PROGRAM Fahrauftrag
VAR
	//State machine
	sStart : BOOL := TRUE;
	s0,s1a,s1b,s2,s3,s4,s5,s6a,s6b,s7,s8,s9,s10,s11a,s11b,s12,s13,s14,s15,s16,s17,s18,s19,s20,s21a,s21b,s22,s23,s24,s25,s26a,s26b,s27,s28,s29,s30,s31: BOOL := FALSE;
	sk0, sk1, sk2, sk3, sk4, sk10, sk20, sk21, sk22, sk23, sk24, sk25, sk26, sk27, sk28, sk29, sk30, sk31 : BOOL := FALSE; //States von Kollision
	
	AStar : AStar;										//A-Stern Algorithmus
	readAssigment: ReadAssigment;						//Auswertung des Auftrags
	TrajectoryController: TrajectoryControl;			//Schnittstelle zu GW3
	
	wayPointList : ARRAY[0..100] OF RobotPoseSimple;	//Wegpunktliste
	actualCamX, actualCamY : LREAL;						//letzte Kameradaten ungleich 0
	lastRelevantStateForCollision : STRING(5);			//letzter State für Rückfall bei Kollision
	
	//Schnittstelle zum MQTT_PRG
	FeedbackToGW1 AT%Q*: STRING(50);		//Feedback/Status des Roboters an GW1
	resetVar, resetGoBack AT%Q*: BOOL;					//messages von MQTT zurücksetzen
	RoboNmbToGoBack AT%Q* : INT;
	Auftrag AT%I*: Auftrag;					//Auftrag von GW1
	StatusFromGW1 AT%I*: STRING(50);		//Status von GW1
	goBack AT%I* : BOOL;					//zurückfahren auf Befehl von anderem HAWino
	reset AT%I* : BOOL;						//Fahrauftrag und GW3 zurücksetzen auf Befehl von GW1
	
	//Schnittstelle zu A*-Algorithmus
	EndNode : INT;							//letzter Knoten
	xEndvalue : LREAL;						//Ziel xKoordinate
	xRobotStartposition : LREAL;			//aktuelle xKoordinate
	yEndvalue : LREAL;						//Ziel yKoordinate
	yRobotStartposition : LREAL;			//aktuelle yKoordinate
	xPointList : ARRAY[0..100] OF LREAL;	//xKoordinatenliste
	yPointList : ARRAY[0..100] OF LREAL;	//yKoordinatenliste
	finished_ASearch : BOOL;	 			//Variable, dass Algorithmus fertig
	i: INT;									//Laufvariable zum Übertragen der x und y Koordinaten in die Wegpunktliste
	zeile: INT;								//Arrayindex, wo Wegpunktliste zuende
	
	//Kollision
	collision AT%I*: ARRAY[0..4] OF BOOL;		//Collision wurde erkannt
	lastCollision: ARRAY [0..4] OF BOOL;		//letzte Collision gespeichert
	collisionFree, collisionSolutionWorking : BOOL;				//keine Kollision aktuell
	removeNodeCollision : ARRAY[1..11] OF INT;	//Nodes die durch anderen HAWino blockiert
	todo : STRING(10);							//Aufgabe von diesem HAWino bei Kollision (fahren oder warten)
	firstTime: BOOL := TRUE;	
	timerCollision : TON;						//Zeit die bei Kollision gewartet wird, bevor Reaktion folgt
	otherRobo : ARRAY[0..4] OF INT;				//andere HAWinos, die an Kollision beteilgit
	otherRoboAtStation, otherRoboAtStop, thisRoboAtStation, drivingAtStation, newCollision : BOOL;			//anderer beteiligter HAWino ist im Stationsbereich
	
	//error
	noCamera, AStarFailed, error, test : BOOL;
	resetTimer : TON;
END_VAR

timerCollision();
resetTimer();
errorTest();

collisionFree := NOT collision[Var_HAWIno.Robot_Number];

//neue Kollision angekommen oder noch alte?
//IF lastCollision[1] <> collision[1] OR lastCollision[2] <> collision[2] OR lastCollision[3] <> collision[3] OR lastCollision[4] <> collision[4] OR collision[0] THEN
//	IF collision[Var_HAWIno.Robot_Number] THEN
//		TrajectoryController.xBoEnable := FALSE;
//		CollisionSolution();
//		timerCollision.IN := TRUE;
//		timerCollision.PT := T#2S;
//	END_IF
//	lastCollision := collision;
//LSIF (todo = 'Warten' AND collisionFree) OR timerCollision.Q THEN
//	CollisionSolution();	
//	timerCollision.IN := FALSE;
//ELSIF (goBack AND NOT resetGoBack) OR (otherRoboAtStation AND todo = 'Warten') THEN
//	drivingBack();
//	todo := 'Warten';
//ELSIF resetGoBack AND NOT goBack THEN
//	resetGoBack := FALSE;
//END_IF

IF lastCollision[1] <> collision[1] OR lastCollision[2] <> collision[2] OR lastCollision[3] <> collision[3] OR lastCollision[4] <> collision[4] OR collision[0] THEN
	newCollision := TRUE;
	lastCollision := collision;
END_IF

IF collision[Var_HAWIno.Robot_Number] AND newCollision THEN
	TrajectoryController.xBoEnable := FALSE;
	IF NOT collisionSolutionWorking THEN
		sk0 := TRUE;
	END_IF
	CollisionsSolution_new();
	newCollision := FALSE;
	timerCollision.IN := TRUE;
	timerCollision.PT := T#2S;
ELSIF collisionSolutionWorking THEN
	CollisionsSolution_new();
END_IF

//Camera damit immer Daten da
IF camera.cameraData.robotPositionArray[Var_HAWIno.Robot_Number].x <> 0 AND camera.cameraData.robotPositionArray[Var_HAWIno.Robot_Number].y <> 0 THEN
	actualCamX := camera.cameraData.robotPositionArray[Var_HAWIno.Robot_Number].x;
	actualCamY := camera.cameraData.robotPositionArray[Var_HAWIno.Robot_Number].y;
END_IF

////////////////////////////////////////////////////////StateMaschine/////////////////////////////////////////////////

//Init
IF sStart AND NOT s0 THEN
	lastRelevantStateForCollision := 's0';
	sStart := 0; s0 := 1;
	//	RückmeldungGW1 Verfügbar
	FeedbackToGW1 := 'Verfuegbar';
	resetVar := FALSE;
	TrajectoryController.xBoReset := FALSE;
END_IF

//////////////////////////////////////////////////////////////////////////////////////////////////////////////
//////////////////////////////////FAHRAUFTRAG/////////////////////////////////////////////////////////////////
//////////////////////////////////////////////////////////////////////////////////////////////////////////////

//	Warten auf Auftrag
IF s0 AND NOT s1a AND Auftrag.Art = 'Fahrauftrag' THEN
	s0 := 0; s1a := 1;
	lastRelevantStateForCollision := 's1a';
	//	RückmeldugGW1 Auftrag angenommen setzt
	FeedbackToGW1 := 'Auftrag angenommen';
	//Auftrag auswerten
	readAssigment(assigment:= Auftrag);
	EndNode := readAssigment.endNodePickup;															
	xEndvalue := readAssigment.pickupLocation.x;
	yEndvalue := readAssigment.pickupLocation.y;
	xRobotStartposition := camera.cameraData.robotPositionArray[Var_HAWIno.Robot_Number].x;
	yRobotStartposition := camera.cameraData.robotPositionArray[Var_HAWIno.Robot_Number].y;	
END_IF

IF s1a AND NOT s1b AND xRobotStartposition <> 0 AND yRobotStartposition <> 0 THEN
	s1a := 0; s1b := 1;
	AStar(xRobotActual := xRobotStartposition, yRobotActual := yRobotStartposition, xEnd := xEndvalue, yEnd := yEndvalue, endNode := EndNode, blockedNodes := removeNodeCollision);
	finished_ASearch := AStar.finishedASearch;
	xPointList := AStar.xCoordinates;
	yPointList := AStar.yCoordinates;
	ZEROS_INT(removeNodeCollision);
ELSIF s1a AND NOT s1b THEN
	xRobotStartposition := actualCamX;
	yRobotStartposition := actualCamY;
END_IF

//Bahnplanung
IF s1b AND NOT s2 AND finished_ASearch THEN
	ZEROS_RobotPoseSimple(wayPointList);
	FOR i := 0 TO 100 BY 1 DO
 		wayPointList[i] := ToRobotPoseSimple(x:= xPointList[i], y:= yPointList[i], theta:= -1);
		IF xPointList[i] = 0 THEN
			zeile := i;
			EXIT;
		END_IF
	END_FOR
	wayPointList[zeile] := readAssigment.pickupLocation;
	wayPointList[zeile+1] := ToRobotPoseSimple(x := -1, y := -1, theta := -1);
	//wayPointList[zeile+2] := readAssigment.lastPointsToPickup[2];
	TrajectoryController.setWaypointList(waypointList);
	trajectoryController.newWaypointListAvailable := TRUE;
	s1b := 0; s2 := 1;
END_IF

///////////////////////////////////////////////FahrtZumAbholort///////////////////////////////////////////////////

// 	RückmeldungGW3 Wegpunkte erhalten abwarten
IF s2 AND NOT s3 AND trajectoryController.yControllerState = ControllerState.setTrajectory THEN
	s2 := 0; s3 := 1;
	trajectoryController.newWaypointListAvailable := FALSE;
END_IF

// 	RückmeldungGW3 ready abwarten
IF s3 AND NOT s4 AND trajectoryController.yControllerState = ControllerState.ready THEN
	s3 := 0; s4 := 1;
	trajectoryController.xBoEnable := TRUE;
END_IF
	
//	RückmeldungGW3 Fahrt abwarten
IF s4 AND NOT s5 AND trajectoryController.yControllerState = ControllerState.driving THEN
	s4 := 0; s5 := 1;
	//	RückmeldungGW1 Auf Anfahrt setzen
	FeedbackToGW1 := 'Auf Anfahrt';
END_IF

//	RückmeldungGW3 am Ziel abwarten
IF s5 AND NOT s6a AND trajectoryController.yBoArrivedAtDestination THEN
	s5 := 0; s6a := 1;
	lastRelevantStateForCollision := 's6a';
	trajectoryController.xBoEnable := FALSE;
	//	Greifersteuerung
	Gripper.closeGripperCommand := TRUE;
END_IF
												// hier könnte noch slider und Lichtschranke abgefragt werden zur Sicherheit
IF s6a AND NOT s6b AND NOT Gripper.partGripped THEN
	s6a := 0; s6b := 1;	
	//	RückmeldungGW1 Teil aufgenommen setzen
	FeedbackToGW1 := 'Teil aufgenommen';
	//	Fahrauftrag zu Lesekopf
	ZEROS_RobotPoseSimple(wayPointList);
	wayPointList := readAssigment.pointsFromSlotToReader;
	TrajectoryController.setWaypointList(wayPointList);
	trajectoryController.newWaypointListAvailable := TRUE;
ELSIF s6a AND NOT s6b AND Gripper.partGripped THEN
	Gripper.closeGripperCommand := FALSE;
	ZEROS_RobotPoseSimple(wayPointList);										//test, sonst für alle
	wayPointList[0] := ToRobotPoseSimple(x := readAssigment.pickupLocation.x - 100, y := readAssigment.pickupLocation.y, theta := readAssigment.pickupLocation.theta);
	wayPointList[1] := readAssigment.pickupLocation;
	wayPointList[2] := ToRobotPoseSimple(x := -1, y := -1, theta := -1);
	TrajectoryController.setWaypointList(waypointList);
	trajectoryController.newWaypointListAvailable := TRUE;
	s6a := 0; s2 := 1;
END_IF


/////////////////////////////////////////////////////FahrtZumLesekopf/////////////////////////////////////////////////////////

// 	RückmeldungGW3 Wegpunkte erhalten abwarten
IF s6b AND NOT s7 AND trajectoryController.yControllerState = ControllerState.setTrajectory AND gripper.state = CoreGripperControlState.Open THEN
	s6b := 0; s7 := 1;
	trajectoryController.newWaypointListAvailable := FALSE;
END_IF

// 	RückmeldungGW3 ready abwarten
IF s7 AND NOT s8 AND trajectoryController.yControllerState = ControllerState.ready THEN
	s7 := 0; s8 := 1;
	trajectoryController.xBoEnable := TRUE;
END_IF
	
//	RückmeldungGW3 Fahrt abwarten
IF s8 AND NOT s9 AND trajectoryController.yControllerState = ControllerState.driving THEN
	s8 := 0; s9 := 1;
END_IF

//	RückmeldungGW3 am Ziel abwarten
IF s9 AND NOT s10 AND trajectoryController.yBoArrivedAtDestination THEN
	s9 := 0; s10 := 1;
	lastRelevantStateForCollision := 's10';
	trajectoryController.xBoEnable := FALSE;
	//	RückmeldungGW1 Abmeldung
	FeedbackToGW1 := 'Abmeldung';
END_IF

//	Warten auf Werkstück ausgelesen
IF s10 AND NOT s11a AND StatusFromGW1 = 'WerkstueckAusgelesen' THEN
	s10 := 0; s11a := 1;
	lastRelevantStateForCollision := 's11a';
	resetVar := TRUE;
	
	//Auftrag auswerten
	EndNode   := readAssigment.endNodeStorage;																	
	xEndvalue := readAssigment.storageLocation.x;
	yEndvalue := readAssigment.storageLocation.y;
	yRobotStartposition := camera.cameraData.robotPositionArray[Var_HAWIno.Robot_Number].y;	
	xRobotStartposition := camera.cameraData.robotPositionArray[Var_HAWIno.Robot_Number].x;
	//IF readAssigment.assigment.AbholTasche < 3 THEN
	//	xRobotStartposition := camera.cameraData.robotPositionArray[Var_HAWIno.Robot_Number].x - 200;
	//ELSE
	//	xRobotStartposition := camera.cameraData.robotPositionArray[Var_HAWIno.Robot_Number].x + 200;
	//END_IF
END_IF

IF s11a AND NOT s11b AND xRobotStartposition <> 0 AND yRobotStartposition <> 0 THEN
	s11a := 0; s11b := 1;
	AStar(xRobotActual := xRobotStartposition, yRobotActual := yRobotStartposition, xEnd := xEndvalue, yEnd := yEndvalue, endNode := EndNode, blockedNodes := removeNodeCollision);
	finished_ASearch := AStar.finishedASearch;
	xPointList := AStar.xCoordinates;
	yPointList := AStar.yCoordinates;
	ZEROS_INT(removeNodeCollision);
ELSIF s11a AND NOT s11b THEN
	//IF readAssigment.assigment.AbholTasche < 3 THEN	
	//	xRobotStartposition := actualCamX - 200;
	//ELSE
	//	xRobotStartposition := actualCamX + 200;
	//END_IF
	xRobotStartposition := actualCamX;
	yRobotStartposition := actualCamY;
END_IF

//Bahnplanung
IF s11b AND NOT s12 AND finished_ASearch THEN
	ZEROS_RobotPoseSimple(wayPointList);
	FOR i := 0 TO 100 BY 1 DO
 		wayPointList[i] := ToRobotPoseSimple(x:= xPointList[i], y:= yPointList[i], theta:= -1);
		IF xPointList[i] = 0 THEN
			zeile := i;
			EXIT;
		END_IF
	END_FOR
	wayPointList[zeile] := readAssigment.readerCheckIn;
	wayPointList[zeile+1] := ToRobotPoseSimple(x := -1, y := -1, theta := -1);
	TrajectoryController.setWaypointList(waypointList);
	trajectoryController.newWaypointListAvailable := TRUE;
	s11b := 0; s12 := 1;
END_IF

/////////////////////////////////////////////////FahrtZurAblageStation///////////////////////////////////////////////////

// 	RückmeldungGW3 Wegpunkte erhalten abwarten
IF s12 AND NOT s13 AND trajectoryController.yControllerState = ControllerState.setTrajectory THEN
	s12 := 0; s13 := 1;
	trajectoryController.newWaypointListAvailable := FALSE;
END_IF

// 	RückmeldungGW3 ready abwarten
IF s13 AND NOT s14 AND trajectoryController.yControllerState = ControllerState.ready THEN
	s13 := 0; s14 := 1;
	trajectoryController.xBoEnable := TRUE;
END_IF
	
//	RückmeldungGW3 Fahrt abwarten
IF s14 AND NOT s15 AND trajectoryController.yControllerState = ControllerState.driving THEN
	s14 := 0; s15 := 1;
	resetVar := FALSE;
	//	RückmeldungGW1 Auf Anfahrt setzen
	FeedbackToGW1 := 'Auf Transport';
END_IF

//	RückmeldungGW3 am Ziel abwarten
IF s15 AND NOT s16 AND trajectoryController.yBoArrivedAtDestination THEN
	s15 := 0; s16 := 1;
	lastRelevantStateForCollision := 's16';	
	trajectoryController.xBoEnable := FALSE;
	//	RückmeldungGW1 Anmeldung
	FeedbackToGW1 := 'Anmeldung';
END_IF

//	Warten auf Werkstück ausgelesen
IF s16 AND NOT s17 AND StatusFromGW1 = 'WerkstueckAusgelesen' THEN
	s16 := 0; s17 := 1;
	lastRelevantStateForCollision := 's17';
	resetVar := TRUE;
	//	Fahrauftrag zur Ablage
	ZEROS_RobotPoseSimple(wayPointList);
	wayPointList := readAssigment.pointsFromReaderToSlot;
	TrajectoryController.setWaypointList(wayPointList);
	trajectoryController.newWaypointListAvailable := TRUE;
END_IF

//////////////////////////////////////////////////FahrtZurAblage///////////////////////////////////////////////////////

// 	RückmeldungGW3 Wegpunkte erhalten abwarten
IF s17 AND NOT s18 AND trajectoryController.yControllerState = ControllerState.setTrajectory THEN
	s17 := 0; s18 := 1;
	trajectoryController.newWaypointListAvailable := FALSE;
END_IF

// 	RückmeldungGW3 ready abwarten
IF s18 AND NOT s19 AND trajectoryController.yControllerState = ControllerState.ready THEN
	s18 := 0; s19 := 1;
	trajectoryController.xBoEnable := TRUE;
END_IF
	
//	RückmeldungGW3 Fahrt abwarten
IF s19 AND NOT s20 AND trajectoryController.yControllerState = ControllerState.driving THEN
	s19 := 0; s20 := 1;
	resetVar := FALSE;
END_IF

//	RückmeldungGW3 am Ziel abwarten
IF s20 AND NOT s21a AND trajectoryController.yBoArrivedAtDestination THEN
	s20 := 0; s21a := 1;
	lastRelevantStateForCollision := 's21a';
	trajectoryController.xBoEnable := FALSE;
	//	Greifersteuerung
	Gripper.closeGripperCommand := FALSE;
	//	RückmeldungGW1 Teil abgelegt
	FeedbackToGW1 := 'Teil abgelegt';
	//	Fahrauftrag zum Parkplatz
	EndNode := readAssigment.endNodeParking[Var_HAWIno.Robot_Number];															//todo in matlab
	xEndvalue := readAssigment.parkingSlots[Var_HAWIno.Robot_Number].x;
	yEndvalue := readAssigment.parkingSlots[Var_HAWIno.Robot_Number].y;
	//IF readAssigment.assigment.AblageTasche < 3 THEN
	//	xRobotStartposition := camera.cameraData.robotPositionArray[Var_HAWIno.Robot_Number].x - 200;
	//ELSE
	//	xRobotStartposition := camera.cameraData.robotPositionArray[Var_HAWIno.Robot_Number].x + 200;
	//END_IF
	xRobotStartposition := camera.cameraData.robotPositionArray[Var_HAWIno.Robot_Number].x;
	yRobotStartposition := camera.cameraData.robotPositionArray[Var_HAWIno.Robot_Number].y;	
END_IF

				
//////////////////////////////////////////////////////////////////////////////////////////////////////////////
///////////////////////////////////////LADEAUFTRAG////////////////////////////////////////////////////////////
//////////////////////////////////////////////////////////////////////////////////////////////////////////////

IF s0 AND NOT s26a AND Auftrag.Art = 'Ladeauftrag' THEN
	s0 := 0; s26a := 1;
	lastRelevantStateForCollision := 's26a';
	//	RückmeldugGW1 Auftrag angenommen setzt
	FeedbackToGW1 := 'Auftrag angenommen';
	//Auftrag auswerten
	readAssigment(assigment:= Auftrag);
	EndNode := readAssigment.endNodeCharging;
	xEndvalue := readAssigment.chargingLocation.x;
	yEndvalue := readAssigment.chargingLocation.y;
	xRobotStartposition := camera.cameraData.robotPositionArray[Var_HAWIno.Robot_Number].x;
	yRobotStartposition := camera.cameraData.robotPositionArray[Var_HAWIno.Robot_Number].y;	
END_IF

IF s26a AND NOT s26b AND xRobotStartposition <> 0 AND yRobotStartposition <> 0 THEN
	s26a := 0; s26b := 1;
	AStar(xRobotActual := xRobotStartposition, yRobotActual := yRobotStartposition, xEnd := xEndvalue, yEnd := yEndvalue, endNode := EndNode, blockedNodes := removeNodeCollision);
	finished_ASearch := AStar.finishedASearch;
	xPointList := AStar.xCoordinates;
	yPointList := AStar.yCoordinates;
	ZEROS_INT(removeNodeCollision);
ELSIF s26a AND NOT s26b THEN
	xRobotStartposition := actualCamX;
	yRobotStartposition := actualCamY;
END_IF

//Bahnplanung
IF s26b AND NOT s27 AND finished_ASearch THEN
	ZEROS_RobotPoseSimple(wayPointList);
	FOR i := 0 TO 100 BY 1 DO
 		wayPointList[i] := ToRobotPoseSimple(x:= xPointList[i], y:= yPointList[i], theta:= -1);
		IF xPointList[i] = 0 THEN
			zeile := i;
			EXIT;
		END_IF
	END_FOR
	wayPointList[zeile] := readAssigment.chargingLocation;
	wayPointList[zeile+1] := ToRobotPoseSimple(x := -1, y := -1, theta := -1);
	TrajectoryController.setWaypointList(waypointList);
	trajectoryController.newWaypointListAvailable := TRUE;
	resetVar := TRUE;															//testen
	s26b := 0; s27 := 1;
END_IF

///////////////////////////////////////////////FahrtZurStation///////////////////////////////////////////////////

// 	RückmeldungGW3 Wegpunkte erhalten abwarten
IF s27 AND NOT s28 AND trajectoryController.yControllerState = ControllerState.setTrajectory THEN
	s27 := 0; s28 := 1;
	trajectoryController.newWaypointListAvailable := FALSE;
END_IF

// 	RückmeldungGW3 ready abwarten
IF s28 AND NOT s29 AND trajectoryController.yControllerState = ControllerState.ready THEN
	s28 := 0; s29 := 1;
	trajectoryController.xBoEnable := TRUE;
END_IF
	
//	RückmeldungGW3 Fahrt abwarten
IF s29 AND NOT s30 AND trajectoryController.yControllerState = ControllerState.driving THEN
	s29 := 0; s30 := 1;
	//	RückmeldungGW1 Auf Anfahrt setzen
	FeedbackToGW1 := 'Auf Anfahrt';
END_IF

//	RückmeldungGW3 am Ziel abwarten
IF s30 AND NOT s31 AND trajectoryController.yBoArrivedAtDestination THEN
	s30 := 0; s31 := 1;
	lastRelevantStateForCollision := 's31';
	trajectoryController.xBoEnable := FALSE;
	resetVar := FALSE;															//testen
	//	RückmeldungGW1 Teil aufgenommen setzen
	FeedbackToGW1 := 'An Ladestation';
END_IF

IF s31 AND NOT s21a AND StatusFromGW1 = 'FertigGeladen' THEN
	s31 := 0; s21a := 1;
	lastRelevantStateForCollision := 's21a';
	//	Fahrauftrag zum Parkplatz
	EndNode := readAssigment.endNodeParking[Var_HAWIno.Robot_Number];															
	xEndvalue := readAssigment.parkingSlots[Var_HAWIno.Robot_Number].x;
	yEndvalue := readAssigment.parkingSlots[Var_HAWIno.Robot_Number].y;
	xRobotStartposition := camera.cameraData.robotPositionArray[Var_HAWIno.Robot_Number].x;
	yRobotStartposition := camera.cameraData.robotPositionArray[Var_HAWIno.Robot_Number].y;	
END_IF


//////////////////////////////////////////////////////////////////////////////////////////////////////////////
///////////////////////////////////////Parkplatzanfahrt///////////////////////////////////////////////////////
//////////////////////////////////////////////////////////////////////////////////////////////////////////////

IF s21a AND NOT s21b AND xRobotStartposition <> 0 AND yRobotStartposition <> 0 AND gripper.state = CoreGripperControlState.Closed THEN
	s21a := 0; s21b := 1;
	AStar(xRobotActual := xRobotStartposition, yRobotActual := yRobotStartposition, xEnd := xEndvalue, yEnd := yEndvalue, endNode := EndNode, blockedNodes := removeNodeCollision);
	finished_ASearch := AStar.finishedASearch;
	xPointList := AStar.xCoordinates;
	yPointList := AStar.yCoordinates;
	ZEROS_INT(removeNodeCollision);
ELSIF s21a AND NOT s21b THEN
	//IF readAssigment.assigment.AbholTasche < 3 THEN	
	//	xRobotStartposition := actualCamX - 200;
	//ELSE
	//	xRobotStartposition := actualCamX + 200;
	//END_IF
	xRobotStartposition := actualCamX;
	yRobotStartposition := actualCamY;
END_IF

//Bahnplanung
IF s21b AND NOT s22 AND finished_ASearch THEN
	ZEROS_RobotPoseSimple(wayPointList);
	FOR i := 0 TO 100 BY 1 DO
 		wayPointList[i] := ToRobotPoseSimple(x:= xPointList[i], y:= yPointList[i], theta:= -1);
		IF xPointList[i] = 0 THEN
			zeile := i;
			EXIT;
		END_IF
	END_FOR
	wayPointList[zeile] := readAssigment.parkingSlots[Var_HAWIno.Robot_Number];
	wayPointList[zeile+1] := ToRobotPoseSimple(x := -1, y := -1, theta := -1);
	TrajectoryController.setWaypointList(waypointList);
	trajectoryController.newWaypointListAvailable := TRUE;
	s21b := 0; s22 := 1;
END_IF


///////////////////////////////////////////////////FahrtZumParkplatz////////////////////////////////////////////////////////
 
// 	RückmeldungGW3 Wegpunkte erhalten abwarten
IF s22 AND NOT s23 AND trajectoryController.yControllerState = ControllerState.setTrajectory THEN
	s22 := 0; s23 := 1;
	trajectoryController.newWaypointListAvailable := FALSE;
END_IF

// 	RückmeldungGW3 ready abwarten
IF s23 AND NOT s24 AND trajectoryController.yControllerState = ControllerState.ready THEN
	s23 := 0; s24 := 1;
	trajectoryController.xBoEnable := TRUE;
END_IF
	
//	RückmeldungGW3 Fahrt abwarten
IF s24 AND NOT s25 AND trajectoryController.yControllerState = ControllerState.driving THEN
	s24 := 0; s25 := 1;
	//kann schon nächsten Auftrag annehmen
	FeedbackToGW1 := 'Verfuegbar';
END_IF

IF s25 AND trajectoryController.yControllerState = ControllerState.driving AND Auftrag.Art = 'Fahrauftrag' THEN
	lastRelevantStateForCollision := 's0';
	trajectoryController.xBoEnable := FALSE;
	s25 := 0; s0 := 1;
END_IF

//	RückmeldungGW3 am Ziel abwarten
IF s25 AND NOT s0 AND trajectoryController.yBoArrivedAtDestination THEN
	s25 := 0; s0 := 1;
	lastRelevantStateForCollision := 's0';
	trajectoryController.xBoEnable := FALSE;
	//	RückmeldungGW1 Verfügbar
	FeedbackToGW1 := 'Verfuegbar';
END_IF

////////////////////////////////////////////////////////RESET/////////////////////////////////////////////////////
IF reset THEN
	TrajectoryController.xBoEnable := FALSE;
	doReset();
	resetTimer.PT := T#1S;
	resetTimer.IN := TRUE;
END_IF

IF Auftrag.Art = '' AND (trajectoryController.yControllerState = ControllerState.idle OR trajectoryController.yControllerState = ControllerState.ready) AND resetTimer.Q THEN
	//reset zurücksetzen
	resetTimer.IN := FALSE;
	reset := FALSE;
	EndNode := readAssigment.endNodeParking[Var_HAWIno.Robot_Number];															//todo in matlab
	xEndvalue := readAssigment.parkingSlots[Var_HAWIno.Robot_Number].x;
	yEndvalue := readAssigment.parkingSlots[Var_HAWIno.Robot_Number].y;
	xRobotStartposition := camera.cameraData.robotPositionArray[Var_HAWIno.Robot_Number].x;
	yRobotStartposition := camera.cameraData.robotPositionArray[Var_HAWIno.Robot_Number].y;	
	s21a := TRUE;
	lastRelevantStateForCollision := 's21a';
	resetVar := FALSE;
	TrajectoryController.xBoReset := FALSE;
END_IF

METHOD CollisionSolution : BOOL
VAR_INPUT
END_VAR
VAR
	//lastCollision : ARRAY[1..5] OF BOOL;
	roboNmb, nmb, n : INT;
	i : INT := 1;
	otherRoboAtStop : BOOL;
	//collisionAtStation: BOOL;
	timeout : BOOL;
END_VAR
//wenn Zielknoten gelöscht wird weil Roboter im Weg steht, dann paar Schritte zurückfahren und dem anderen Platz machen...

IF NOT collisionFree AND NOT timerCollision.Q THEN
	//gestoppt
	//alle States zurücknehmen
	removeAllToken();
	i := 0;
		
	//rausfinden welche Roboter beteiligt
	FOR nmb := 0 TO 4 BY 1 DO
		IF collision[nmb] AND nmb <> Var_HAWIno.Robot_Number THEN
			otherRobo[i] := nmb;
			i := i + 1;
		END_IF
	END_FOR
	
	todo := 'Warten';
	//darf ich fahren? nur wenn kleinere Roboternummer
	FOR n := 0 TO 4 BY 1 DO
		IF otherRobo[n] > Var_HAWIno.Robot_Number THEN
			todo := 'Fahren';
		END_IF
	END_FOR
	
	IF otherRobo[0] > 0 THEN
		IF camera.cameraData.robotPositionArray[otherRobo[0]].x = 0 AND camera.cameraData.robotPositionArray[otherRobo[0]].x = 0 THEN
			noCamera := TRUE; //sinnvoll?????
		ELSIF camera.cameraData.robotPositionArray[otherRobo[0]].x > 7000 AND camera.cameraData.robotPositionArray[otherRobo[0]].x < 7200  THEN
			//Anderer Roboter auf Parkplatz
			otherRoboAtStop := TRUE;	
		ELSIF camera.cameraData.robotPositionArray[otherRobo[0]].x > 6100 AND camera.cameraData.robotPositionArray[otherRobo[0]].x < 6800 AND camera.cameraData.robotPositionArray[otherRobo[0]].y > 3400 AND camera.cameraData.robotPositionArray[otherRobo[0]].y < 3600  THEN
			//Anderer Roboter an Ladestation
			otherRoboAtStop := TRUE;
		ELSIF camera.cameraData.robotPositionArray[otherRobo[0]].x > 600 AND camera.cameraData.robotPositionArray[otherRobo[0]].x < 5200 AND camera.cameraData.robotPositionArray[otherRobo[0]].y > 2400 AND camera.cameraData.robotPositionArray[otherRobo[0]].y < 3200  THEN
			//Anderer Roboter im Bereich der Stationen
			otherRoboAtStation := TRUE;
		END_IF
		
		//Stationsfahrt: anderen Robo wegschicken -> Timer nötig????
		IF lastRelevantStateForCollision = 's6a' OR lastRelevantStateForCollision = 's10' OR lastRelevantStateForCollision = 's16' OR lastRelevantStateForCollision = 's17' THEN
			//anderen Wegschicken
			RoboNmbToGoBack := otherRobo[0];
			todo := 'Fahren';
		END_IF
	END_IF
END_IF


IF timerCollision.Q OR collisionFree OR otherRoboAtStop THEN
//warten auf Timer??? - in allen fällen
	RoboNmbToGoBack := 0;
	//höhrer Priorität
	IF todo = 'Fahren' THEN
		//update removeNode - nur wenn nicht an Station
		IF NOT otherRoboAtStation THEN
			findNodesToRemove(collisionRobo := otherRobo);
		END_IF
		
		//in richtigen State zurück zum neuplanen und weiterfahren
		xRobotStartposition := camera.cameraData.robotPositionArray[Var_HAWIno.Robot_Number].x;
		yRobotStartposition := camera.cameraData.robotPositionArray[Var_HAWIno.Robot_Number].y;	
		continueAfterCollision();
		todo := '';
		
	ELSIF todo = 'Warten' THEN
		IF collisionFree OR otherRoboAtStop THEN
			xRobotStartposition := camera.cameraData.robotPositionArray[Var_HAWIno.Robot_Number].x;
			yRobotStartposition := camera.cameraData.robotPositionArray[Var_HAWIno.Robot_Number].y;	
			continueAfterCollision();
			todo := '';
		//ELSIF goback THEN
			//drivingBack();
		END_IF
	END_IF
	timerCollision.IN := FALSE;
END_IF
END_METHOD

METHOD CollisionsSolution_new : BOOL
VAR_INPUT
END_VAR
VAR
	n : INT;
END_VAR
otherRoboInfo();
collisionSolutionWorking := TRUE;
/////////////////////////////////////////////////////////////////NORMAL////////////////////////////////////////////////////////////////////////

IF sk0 AND NOT sk1 AND NOT otherRoboAtStation AND NOT thisRoboAtStation AND NOT otherRoboAtStop AND timerCollision.Q THEN
	todo := 'Warten';
	//darf ich fahren? nur wenn kleinere Roboternummer
	FOR n := 0 TO 4 BY 1 DO
		IF otherRobo[n] > Var_HAWIno.Robot_Number THEN
			todo := 'Fahren';
		END_IF
	END_FOR
	sk0 := 0; sk1 := 1;
	timerCollision.IN := FALSE;
END_IF

IF sk1 AND NOT sk2 AND todo = 'Fahren' THEN
	findNodesToRemove(collisionRobo := otherRobo);
	
	//in richtigen State zurück zum neuplanen und weiterfahren
	xRobotStartposition := camera.cameraData.robotPositionArray[Var_HAWIno.Robot_Number].x;
	yRobotStartposition := camera.cameraData.robotPositionArray[Var_HAWIno.Robot_Number].y;	
	continueAfterCollision();
	todo := '';
	sk1 := 0; sk2 := 1;
END_IF

IF sk1 AND NOT sk3 AND todo = 'Warten' THEN
	sk1 := 0; sk3 := 1;
END_IF

IF sk3 AND NOT sk4 AND collisionFree THEN
	xRobotStartposition := camera.cameraData.robotPositionArray[Var_HAWIno.Robot_Number].x;
	yRobotStartposition := camera.cameraData.robotPositionArray[Var_HAWIno.Robot_Number].y;
	continueAfterCollision();
	todo := '';
	sk3 := 0; sk4 := 1;
END_IF

IF sk2 OR sk4 THEN
	sk2 := 0; sk4 := 0; 
	resetCollision();
END_IF


/////////////////////////////////////////////////////////////ATSTOP////////////////////////////////////////////////////////////////////////////

IF sk0 AND NOT sk10 AND otherRoboAtStop AND timerCollision.Q THEN
	xRobotStartposition := camera.cameraData.robotPositionArray[Var_HAWIno.Robot_Number].x;
	yRobotStartposition := camera.cameraData.robotPositionArray[Var_HAWIno.Robot_Number].y;
	continueAfterCollision();
	timerCollision.IN := FALSE;
	sk0 := 0; sk10 := 1;
END_IF

IF sk10 THEN
	sk10 := 0;
	resetCollision();
END_IF


//////////////////////////////////////////////////////////////ATSTATION///////////////////////////////////////////////////////////////////////////

IF sk0 AND NOT sk20 AND otherRoboAtStation AND NOT thisRoboAtStation AND timerCollision.Q THEN
	sk0 := 0; sk20 := 1;
	timerCollision.IN := FALSE;
END_IF

//nur anderer Robo an Station
IF sk20 AND NOT sk21 AND otherRoboAtStation AND NOT thisRoboAtStation THEN
	sk20 := 0; sk21 := 1;
	//zurückfahren??? - nein erstmal
END_IF

IF sk21 AND NOT sk22 AND NOT otherRoboAtStation THEN
	xRobotStartposition := camera.cameraData.robotPositionArray[Var_HAWIno.Robot_Number].x;
	yRobotStartposition := camera.cameraData.robotPositionArray[Var_HAWIno.Robot_Number].y;
	continueAfterCollision();
	sk21 := 0; sk22 := 1;
END_IF

//
IF sk20 AND NOT sk23 AND NOT otherRoboAtStation AND thisRoboAtStation THEN
	findNodesToRemove(collisionRobo := otherRobo);
	
	//in richtigen State zurück zum neuplanen und weiterfahren
	xRobotStartposition := camera.cameraData.robotPositionArray[Var_HAWIno.Robot_Number].x;
	yRobotStartposition := camera.cameraData.robotPositionArray[Var_HAWIno.Robot_Number].y;	
	continueAfterCollision();
	sk20 := 0; sk23 := 1;
END_IF

//beide an Station
IF sk20 AND NOT sk24 AND otherRoboAtStation AND thisRoboAtStation THEN
	sk20 := 0; sk24 := 1;
END_IF

//dieser Robo auf Transport an Station
IF sk24 AND NOT sk25 AND drivingAtStation THEN
	xRobotStartposition := camera.cameraData.robotPositionArray[Var_HAWIno.Robot_Number].x;
	yRobotStartposition := camera.cameraData.robotPositionArray[Var_HAWIno.Robot_Number].y;	
	continueAfterCollision();
	sk24 := 0; sk25 := 1;
END_IF

//dieser nicht aber anderer auf Transport an Station
IF sk24 AND NOT sk26 AND NOT drivingAtStation AND goBack THEN
	drivingBack();
	IF resetGoBack THEN
		sk24 := 0; sk26 := 1;
	END_IF
END_IF

IF sk26 AND NOT sk27 AND NOT otherRoboAtStation THEN
	xRobotStartposition := camera.cameraData.robotPositionArray[Var_HAWIno.Robot_Number].x;
	yRobotStartposition := camera.cameraData.robotPositionArray[Var_HAWIno.Robot_Number].y;	
	continueAfterCollision();
	sk26 := 0; sk27 := 1;
END_IF

//beide im Stationsbereich und keiner auf Transport an Station
IF sk24 AND NOT sk28 AND NOT drivingAtStation AND NOT goBack THEN
	todo := 'Warten';
	//darf ich fahren? nur wenn kleinere Roboternummer
	FOR n := 0 TO 4 BY 1 DO
		IF otherRobo[n] > Var_HAWIno.Robot_Number THEN
			todo := 'Fahren';
		END_IF
	END_FOR
	sk24 := 0; sk28 := 1;
END_IF

IF sk28 AND NOT sk29 AND todo = 'Fahren' THEN
	xRobotStartposition := camera.cameraData.robotPositionArray[Var_HAWIno.Robot_Number].x;
	yRobotStartposition := camera.cameraData.robotPositionArray[Var_HAWIno.Robot_Number].y;	
	continueAfterCollision();
	sk28 := 0; sk29 := 1;
END_IF

IF sk28 AND NOT sk30 AND todo = 'Warten' THEN
	drivingBack();
	IF resetGoBack THEN
		sk28 := 0; sk30 := 1;
	END_IF
END_IF

IF sk30 AND NOT sk31 AND NOT otherRoboAtStation THEN
	xRobotStartposition := camera.cameraData.robotPositionArray[Var_HAWIno.Robot_Number].x;
	yRobotStartposition := camera.cameraData.robotPositionArray[Var_HAWIno.Robot_Number].y;	
	continueAfterCollision();
	sk30 := 0; sk31 := 1;
END_IF

IF resetGoBack AND NOT goBack THEN
	resetGoBack := FALSE;
END_IF

/////////////////////////////////////////Am Ende der Kollisionsauflösung//////////////////////////////////////////////
IF sk22 OR sk23 OR sk25 OR sk27 OR sk29 OR sk31 THEN
	sk22 := 0; sk23 := 0; sk25 := 0; sk27 := 0; sk29 := 0; sk31 := 0;
	resetCollision();
END_IF
END_METHOD

METHOD continueAfterCollision : BOOL
VAR_INPUT
END_VAR
VAR
	diffToList : ARRAY[0..100] OF LREAL;
	sortedDiff : ARRAY[0..100,1..2] OF LREAL;
	nextIndex, j, n, l, i : INT;
	nullSortedDiff : ARRAY[0..100,1..2] OF LREAL := [202(0)];
END_VAR
IF lastRelevantStateForCollision = 's0' THEN
	s0 := 1;
ELSIF lastRelevantStateForCollision = 's1a' THEN
	s1a := 1;
ELSIF lastRelevantStateForCollision = 's6a' THEN
	s6b := 1;
	//readAssigment.pointsFromSlotToReader
	//Arrays resetten
	ZEROS(diffToList);
	sortedDiff := nullSortedDiff;
	
	FOR i := 0 TO 10 BY 1 DO
		IF readAssigment.pointsFromSlotToReader[i].x > 0 AND readAssigment.pointsFromSlotToReader[i].y > 0 THEN
			//Abstände Roboter zu Wegpunkten
			diffToList[i] := SQRT(EXPT(camera.cameraData.robotPositionArray[Var_HAWIno.Robot_Number].x - readAssigment.pointsFromSlotToReader[i].x,2) + EXPT(camera.cameraData.robotPositionArray[Var_HAWIno.Robot_Number].y - readAssigment.pointsFromSlotToReader[i].y,2));
			FOR n := 0 TO 10 BY 1 DO
				IF diffToList[i] < sortedDiff[n,2] THEN
					FOR l := 9 TO n BY -1 DO
						sortedDiff[l+1,1] := sortedDiff[l,1];
						sortedDiff[l+1,2] := sortedDiff[l,2];
					END_FOR
					sortedDiff[n,2] := diffToList[i];
					sortedDiff[n,1] := i;
					EXIT;
				ELSIF i = 0 THEN
					sortedDiff[0,2] := diffToList[0];
					sortedDiff[0,1] := 0;
					EXIT;
				END_IF
			END_FOR
		END_IF	
	END_FOR
	
	ZEROS_RobotPoseSimple(wayPointList);
	nextIndex := LREAL_TO_INT(MAX(sortedDiff[0,1],sortedDiff[1,1]));
	
	FOR i := 0 TO 100 - nextIndex BY 1 DO 
		wayPointList[i] := readAssigment.pointsFromSlotToReader[nextIndex + i];
	END_FOR 
	TrajectoryController.setWaypointList(wayPointList);
	trajectoryController.newWaypointListAvailable := TRUE;
	
ELSIF lastRelevantStateForCollision = 's10' THEN
	s10 := 1;
ELSIF lastRelevantStateForCollision = 's11a' THEN
	s11a := 1;
ELSIF lastRelevantStateForCollision = 's16' THEN
	s16 := 1;
ELSIF lastRelevantStateForCollision = 's17' THEN
	s17 := 1;
	//readAssigment.pointsFromReaderToSlot
	//Arrays resetten
	ZEROS(diffToList);
	sortedDiff := nullSortedDiff;
	
	FOR i := 0 TO 10 BY 1 DO
		IF readAssigment.pointsFromReaderToSlot[i].x <> 0 AND readAssigment.pointsFromReaderToSlot[i].y <> -1 THEN
			//Abstände Roboter zu Wegpunkten
			diffToList[i] := SQRT(EXPT(camera.cameraData.robotPositionArray[Var_HAWIno.Robot_Number].x - readAssigment.pointsFromReaderToSlot[i].x,2) + EXPT(camera.cameraData.robotPositionArray[Var_HAWIno.Robot_Number].y - readAssigment.pointsFromReaderToSlot[i].y,2));
			FOR n := 0 TO 10 BY 1 DO
				IF diffToList[i] < sortedDiff[n,2] THEN
					FOR l := 9 TO n BY -1 DO
						sortedDiff[l+1,1] := sortedDiff[l,1];
						sortedDiff[l+1,2] := sortedDiff[l,2];
					END_FOR
					sortedDiff[n,2] := diffToList[i];
					sortedDiff[n,1] := i;
					EXIT;
				ELSIF i = 0 THEN
					sortedDiff[0,2] := diffToList[0];
					sortedDiff[0,1] := 0;
					EXIT;
				END_IF
			END_FOR
		END_IF	
	END_FOR
	
	ZEROS_RobotPoseSimple(wayPointList);
	nextIndex := LREAL_TO_INT(MAX(sortedDiff[0,1],sortedDiff[1,1]));
	
	FOR i := 0 TO 100 - nextIndex BY 1 DO 
		wayPointList[i] := readAssigment.pointsFromReaderToSlot[nextIndex + i];
	END_FOR 
	TrajectoryController.setWaypointList(wayPointList);
	trajectoryController.newWaypointListAvailable := TRUE;
	
ELSIF lastRelevantStateForCollision = 's21a' THEN
	s21a := 1;
ELSIF lastRelevantStateForCollision = 's26a' THEN
	s26a := 1;
ELSIF lastRelevantStateForCollision = 's31' THEN
	s31 := 1;
END_IF
END_METHOD

METHOD doReset : BOOL
VAR_INPUT
END_VAR
resetVar := TRUE;
TrajectoryController.xBoReset := TRUE;
ZEROS_RobotPoseSimple(wayPointList);
actualCamX := 0;
actualCamY := 0;
trajectoryController.newWaypointListAvailable := FALSE;
trajectoryController.xBoEnable := FALSE;
FeedbackToGW1 := 'Verfuegbar';
Gripper.closeGripperCommand := FALSE;
ZEROS_INT(removeNodeCollision);
error := FALSE;

//Statemaschine zurücksetzen
sStart := FALSE;
s0 := FALSE;
s1a := FALSE;
s1b := FALSE;
s2 := FALSE;
s3 := FALSE;
s4 := FALSE;
s5 := FALSE;
s6a := FALSE;
s6b := FALSE;
s7 := FALSE;
s8 := FALSE;
s9 := FALSE;
s10 := FALSE;
s11a := FALSE;
s11b := FALSE;
s12 := FALSE;
s13 := FALSE;
s14 := FALSE;
s15 := FALSE;
s16 := FALSE;
s17 := FALSE;
s18 := FALSE;
s19 := FALSE;
s20 := FALSE;
s21a := FALSE;
s21b := FALSE;
s22 := FALSE;
s23 := FALSE;
s24 := FALSE;
s25 := FALSE;
s26a := FALSE;
s26b := FALSE;
s27 := FALSE;
s28 := FALSE;
s29 := FALSE;
s30 := FALSE;
s31 := FALSE;

resetCollision();
END_METHOD

METHOD drivingBack : BOOL
VAR_INPUT
END_VAR

VAR
	gbWayPointList : ARRAY[0..100] OF RobotPoseSimple;
	diffToList : ARRAY[0..100] OF LREAL;
	sortedDiff : ARRAY[0..100,1..2] OF LREAL;
	index, n, l, i : INT;
	camX, camY : LREAL;
	alternativeGoAway: BOOL;
	nullSortedDiff : ARRAY[0..100,1..2] OF LREAL := [202(0)];
END_VAR
IF firstTime THEN //hier and goBack entfernt
	//Arrays resetten
	ZEROS_RobotPoseSimple(gbWayPointList);
	ZEROS(diffToList);
	sortedDiff := nullSortedDiff;
	alternativeGoAway := FALSE;

	camX := camera.cameraData.robotPositionArray[Var_HAWIno.Robot_Number].x;
	camY := camera.cameraData.robotPositionArray[Var_HAWIno.Robot_Number].y;
	IF camX = 0 AND camY = 0 THEN
		camX := actualCamX;
		camY := actualCamY;
	END_IF
	
	FOR i := 0 TO 100 BY 1 DO
		IF wayPointList[i].x <> 0 AND wayPointList[i].y <> 0 THEN
			//Abstände Roboter zu Wegpunkten
			diffToList[i] := SQRT(EXPT(camX - wayPointList[i].x,2) + EXPT(camY - wayPointList[i].y,2));
			FOR n := 0 TO 100 BY 1 DO
				IF diffToList[i] < sortedDiff[n,2] THEN
					FOR l := 99 TO n BY -1 DO
						sortedDiff[l+1,1] := sortedDiff[l,1];
						sortedDiff[l+1,2] := sortedDiff[l,2];
					END_FOR
					sortedDiff[n,2] := diffToList[i];
					sortedDiff[n,1] := i;
					EXIT;
				ELSIF i = 0 THEN
					sortedDiff[0,2] := diffToList[0];
					sortedDiff[0,1] := 0;
					EXIT;
				ELSIF sortedDiff[n+1,2] = 0 THEN
					sortedDiff[n+1,2] := diffToList[i];
					sortedDiff[n+1,1] := i;
					EXIT;
				END_IF
			END_FOR
		END_IF	
	END_FOR
	
	index := LREAL_TO_INT(MIN(sortedDiff[0,1],sortedDiff[1,1]));

	IF index > 1 THEN
		gbWaypointList[0] := wayPointList[index];
		gbWaypointList[1] := wayPointList[index-1];
		gbWaypointList[2] := wayPointList[index-2];
		gbWaypointList[3] := ToRobotPoseSimple(x := -1, y := -1, theta := -1);
	ELSE
		alternativeGoAway := TRUE;
	END_IF
	
	TrajectoryController.setWaypointList(gbWaypointList);
	trajectoryController.newWaypointListAvailable := TRUE;
	firstTime := FALSE;
END_IF

IF trajectoryController.yControllerState = ControllerState.setTrajectory THEN //hier and goBack entfernt
	trajectoryController.newWaypointListAvailable := FALSE;
END_IF

// 	RückmeldungGW3 ready abwarten
IF trajectoryController.yControllerState = ControllerState.ready THEN //hier and goBack entfernt
	trajectoryController.xBoEnable := TRUE;
END_IF

IF trajectoryController.yBoArrivedAtDestination THEN //hier and goBack entfernt
	trajectoryController.xBoEnable := FALSE;
	resetGoBack := true;
	firstTime := TRUE;
	otherRoboAtStation := FALSE;
END_IF
END_METHOD

METHOD errorTest : BOOL
VAR_INPUT
END_VAR
//ERROR: Teil verloren
IF gripper.state = CoreGripperControlState.Open AND Gripper.partGripped THEN
	error := TRUE;
	TrajectoryController.xBoEnable := FALSE;	
	removeAllToken();
	FeedbackToGW1 := 'Error Teil verloren';
	Gripper.closeGripperCommand := FALSE;
END_IF

//ERROR: Error von GW3
IF trajectoryController.yControllerState = ControllerState.error THEN
	error := TRUE;
	removeAllToken();
	FeedbackToGW1 := 'Error GW3';
	Gripper.closeGripperCommand := FALSE;
END_IF
END_METHOD

METHOD findNodesToRemove : BOOL
VAR_INPUT
	collisionRobo : ARRAY[0..4] OF INT;
END_VAR
VAR
	xMinBox, xMaxBox, yMinBox, yMaxBox, row, col : LREAL;
	xNode, yNode : ARRAY[1..170] OF LREAL;
	d, j, w : INT;
END_VAR
//abfangen wenn keine Kameradaten da?
w := 1;

FOR d := 0 TO 4 BY 1 DO
	IF collisionRobo[d] <> 0 THEN
		//Umrechnung von Knoten in Koordinaten
		 row := 600;
		 col := 200;
		 
		 FOR i := 1 TO 144 BY 1 DO
			 IF xNode[i] <> 10000 THEN
				xNode[i] := col;
			 END_IF
			 IF yNode[i] <> 10000 THEN
				yNode[i] := row;
			 END_IF
			 col := col + 400;
			 IF i MOD 18 = 0 THEN
				 col := 200;
				 row := row + 400;
			 END_IF
		 END_FOR
		 
		 xNode[145] := 850;
		 xNode[146] := 850;
		 xNode[147] := 850;
		 xNode[148] := 1350;
		 xNode[149] := 1350;
		 xNode[150] := 1350;
		 xNode[151] := 2050;
		 xNode[152] := 2050;
		 xNode[153] := 2050;
		 xNode[154] := 2490;
		 xNode[155] := 2490;
		 xNode[156] := 2490;
		 xNode[157] := 3190;
		 xNode[158] := 3190;
		 xNode[159] := 3190;
		 xNode[160] := 3700;
		 xNode[161] := 3700;
		 xNode[162] := 3700;
		 xNode[163] := 4420;
		 xNode[164] := 4420;
		 xNode[165] := 4420;
		 xNode[166] := 4940;
		 xNode[167] := 4940;
		 xNode[168] := 4940;
		 xNode[169] := 6117;
		 xNode[170] := 6716;
		 
		 yNode[145] := 2735;
		 yNode[146] := 2838;
		 yNode[147] := 2936;
		 yNode[148] := 2736;
		 yNode[149] := 2835;
		 yNode[150] := 2935;
		 yNode[151] := 2731;
		 yNode[152] := 2829;
		 yNode[153] := 2931;
		 yNode[154] := 2732;
		 yNode[155] := 2833;
		 yNode[156] := 2928;
		 yNode[157] := 2732;
		 yNode[158] := 2837;
		 yNode[159] := 2940;
		 yNode[160] := 2732;
		 yNode[161] := 2840;
		 yNode[162] := 2940;
		 yNode[163] := 2732;
		 yNode[164] := 2838;
		 yNode[165] := 2944;
		 yNode[166] := 2746;
		 yNode[167] := 2855;
		 yNode[168] := 2942;
		 yNode[169] := 3450;
		 yNode[170] := 3450;
		 
		
		//im Abstand von 400 all Knoten um robot löschen
		xMinBox := camera.cameraData.robotPositionArray[collisionRobo[d]].x - 400;
		xMaxBox := camera.cameraData.robotPositionArray[collisionRobo[d]].x + 400;
		yMinBox := camera.cameraData.robotPositionArray[collisionRobo[d]].y - 400;
		yMaxBox := camera.cameraData.robotPositionArray[collisionRobo[d]].y + 400;
		
		FOR j := 1 TO 170 BY 1 DO
			IF xNode[j] > xMinBox AND xNode[j] < xMaxBox AND yNode[j] > yMinBox AND yNode[j] < yMaxBox THEN
				removeNodeCollision[w] := j;
				w := w + 1;
			END_IF
		END_FOR
	END_IF
END_FOR
END_METHOD

METHOD otherRoboInfo : BOOL
VAR_INPUT
END_VAR
VAR
	nmb: INT;
END_VAR
IF newCollision THEN
	removeAllToken();
	i := 0;
	FOR nmb := 0 TO 4 BY 1 DO
		IF collision[nmb] AND nmb <> Var_HAWIno.Robot_Number THEN
			otherRobo[i] := nmb;
			i := i + 1;
		END_IF
	END_FOR
END_IF

IF otherRobo[0] > 0 THEN
	IF camera.cameraData.robotPositionArray[otherRobo[0]].x > 7000 AND camera.cameraData.robotPositionArray[otherRobo[0]].x < 7200  THEN
		//Anderer Roboter auf Parkplatz
		otherRoboAtStop := TRUE;	
	ELSIF camera.cameraData.robotPositionArray[otherRobo[0]].x > 6100 AND camera.cameraData.robotPositionArray[otherRobo[0]].x < 6800 AND camera.cameraData.robotPositionArray[otherRobo[0]].y > 3400 AND camera.cameraData.robotPositionArray[otherRobo[0]].y < 3600  THEN
		//Anderer Roboter an Ladestation
		otherRoboAtStop := TRUE;
	ELSE
		otherRoboAtStop := FALSE;
	END_IF
	
	IF camera.cameraData.robotPositionArray[otherRobo[0]].x > 600 AND camera.cameraData.robotPositionArray[otherRobo[0]].x < 5200 AND camera.cameraData.robotPositionArray[otherRobo[0]].y > 2400 AND camera.cameraData.robotPositionArray[otherRobo[0]].y < 3200  THEN
		//Anderer Roboter im Bereich der Stationen
		otherRoboAtStation := TRUE;
	ELSE
		otherRoboAtStation := FALSE;
	END_IF
	
	IF camera.cameraData.robotPositionArray[Var_HAWIno.Robot_Number].x > 600 AND camera.cameraData.robotPositionArray[Var_HAWIno.Robot_Number].x < 5200 AND camera.cameraData.robotPositionArray[Var_HAWIno.Robot_Number].y > 2400 AND camera.cameraData.robotPositionArray[Var_HAWIno.Robot_Number].y < 3200  THEN
		thisRoboAtStation := TRUE;
	ELSE
		thisRoboAtStation := FALSE;
	END_IF
	
	//Stationsfahrt: anderen Robo wegschicken -> Timer nötig????
	IF lastRelevantStateForCollision = 's6a' OR lastRelevantStateForCollision = 's10' OR lastRelevantStateForCollision = 's16' OR lastRelevantStateForCollision = 's17' THEN
		//anderen Wegschicken
		IF newCollision THEN
			RoboNmbToGoBack := otherRobo[0];
		ELSE
			RoboNmbToGoBack := 0;
		END_IF 
		drivingAtStation := TRUE;
	else
		drivingAtStation := FALSE;
	END_IF
ELSE
	error := TRUE;
	removeAllToken();
END_IF
END_METHOD

METHOD removeAllToken : BOOL
VAR_INPUT
END_VAR
//Statemaschine zurücksetzen
sStart := FALSE;
s0 := FALSE;
s1a := FALSE;
s1b := FALSE;
s2 := FALSE;
s3 := FALSE;
s4 := FALSE;
s5 := FALSE;
s6a := FALSE;
s6b := FALSE;
s7 := FALSE;
s8 := FALSE;
s9 := FALSE;
s10 := FALSE;
s11a := FALSE;
s11b := FALSE;
s12 := FALSE;
s13 := FALSE;
s14 := FALSE;
s15 := FALSE;
s16 := FALSE;
s17 := FALSE;
s18 := FALSE;
s19 := FALSE;
s20 := FALSE;
s21a := FALSE;
s21b := FALSE;
s22 := FALSE;
s23 := FALSE;
s24 := FALSE;
s25 := FALSE;
s26a := FALSE;
s26b := FALSE;
s27 := FALSE;
s28 := FALSE;
s29 := FALSE;
s30 := FALSE;
s31 := FALSE;
END_METHOD

METHOD resetCollision : BOOL
VAR_INPUT
END_VAR
collisionSolutionWorking := FALSE; //Kollision behoben

Zeros_INT(otherRobo);
otherRoboAtStop := FALSE;
otherRoboAtStation := FALSE;
thisRoboAtStation := FALSE;
RoboNmbToGoBack := 0;
drivingAtStation := FALSE;
todo := '';

sk0 := FALSE;
sk1 := FALSE;
sk2 := FALSE;
sk3 := FALSE;
sk4 := FALSE;
sk10 := FALSE;
sk20 := FALSE;
sk21 := FALSE;
sk22 := FALSE;
sk23 := FALSE;
sk24 := FALSE;
sk25 := FALSE;
sk26 := FALSE;
sk27 := FALSE;
sk28 := FALSE;
sk29 := FALSE;
sk30 := FALSE;
sk31 := FALSE;
END_METHOD

END_PROGRAM

(* stored: Version 1.1.0.1, ProductVersion 3.1.4024.11
   POU Fahrauftrag: Id {d11e2ac1-1df3-4b17-bdc0-8c45421bbbdd}, SpecialFunc None
   Method CollisionSolution: Id {4b28bc3d-12ae-4013-b4ca-5ace32b6b8ab}
   Method CollisionsSolution_new: Id {b549cdcd-badb-48a4-b744-c413f414dadb}
   Method continueAfterCollision: Id {bdb23939-8772-4122-86ab-be757c2f916b}
   Method doReset: Id {11fc1a94-8006-4f54-bbc3-6cfe2505c8b8}
   Method drivingBack: Id {62bdf92e-d532-4d8c-b162-66ce008d6195}
   Method errorTest: Id {e469cc9c-ca1f-4674-b1dd-16db9e33a62d}
   Method findNodesToRemove: Id {ef8384d2-b9d5-47a0-af76-48b877d17d18}
   Method otherRoboInfo: Id {e2679d78-4ec4-4c4f-a55e-7f22b5fbb268}
   Method removeAllToken: Id {ae306339-8136-4758-9f9e-43c55251323b}
   Method resetCollision: Id {55e9b937-ae96-4a1c-b254-a88952f35d6c} *)
